(* PLC project Unnamed, Unknown Unnamed 1 *)
(* stored: creationDateTime 2020-11-15T01:01:23, modificationDateTime 2020-11-15T01:01:23 *)

CONFIGURATION Config0
  RESOURCE Res0 ON PLC
  END_RESOURCE
END_CONFIGURATION
